TYPE ST_SPM_HMI_04 :
STRUCT
	bDaneUtworzone			: BOOL;
	refarrTryby				: REFERENCE TO ARRAY [0..GVL_MachineControlConstans.COUNT_OPERATION_MODES] OF ITF_SITP_Element;
	refArrPoleceniaTrybu	: REFERENCE TO ARRAY [0..GVL_MachineControlConstans.COUNT_MODE_COMMANDS] OF ITF_SITP_PolecenieZmianyTrybu;
END_STRUCT
END_TYPE

(* stored: Version 1.1.0.1
   DUT ST_SPM_HMI_04: Id {74343da3-220d-0ee2-0053-531c3dd2b6a4} *)
